// TwinCAT 3 PLC project Nepionic_Log_OTel
// Title: Nepionic_Log_OTel
// Company: Nepionic
// Author: Nepionic
// ProjectVersion: 0.1.0
// ProgramVersion: 3.1.4026.21
// libraries:
//   [Nepionic_Log], * (Nepionic)
//   Tc2_System, * (Beckhoff Automation GmbH)
//   Tc2_Utilities, * (Beckhoff Automation GmbH)
// project tree:
//   Lib/ OTelLogAppender.TcPOU, OTelLogEntry.TcDUT, OTelLogRing.TcDUT

// ---- Lib/OTelLogEntry.TcDUT
// One slot in the OTelLogRing.
//
// Binary layout (1280 bytes, little-endian, matches Go parser in adsbridge/ringbuf.go):
//
//   offset    0  ULINT   timestamp         Unix epoch nanoseconds
//   offset    8  UDINT   severity          0=Debug 1=Info 2=Warning 3=Error 4=Fatal
//   offset   12  UDINT   attr_count        Number of populated entries in attrs (0..10)
//   offset   16  BYTE[192] message         STRING(191) null-terminated
//   offset  208  BYTE[64]  source          STRING(63)  null-terminated (instance path)
//   offset  272  BYTE[960] attrs           ARRAY[0..9] OF LogAttribute (96 bytes each)
//                                            each attr:
//                                              offset  0  key         STRING(31)       = 32 bytes
//                                              offset 32  attr_type   LogAttributeType =  1 byte
//                                              offset 33  value_bytes ARRAY[0..62]     = 63 bytes
//   offset 1232  BYTE[44]  _pad
//   offset 1276  UDINT   sequence          ODD=being written, EVEN=committed (LAST field)
//   Total: 1280 bytes
{attribute 'pack_mode' := '1'}
TYPE OTelLogEntry :
STRUCT
	timestamp : ULINT;
	severity : UDINT;
	attribute_count : UDINT(0..10);
	message : STRING(191);
	source : STRING(63);
	attributes : ARRAY[0..9] OF Nepionic_Log.LogAttribute;
	_pad : ARRAY[0..43] OF BYTE;
	sequence : UDINT;
END_STRUCT
END_TYPE

// ---- Lib/OTelLogRing.TcDUT
// Ring buffer header + 128-slot log entry array.
// Exposed as an ADS symbol (e.g. OtelBridge.LogRing) and read by the Go collector.
//
// Binary layout:
//   offset  0  UDINT  head          Monotonically increasing write counter
//   offset  4  UDINT  capacity      Number of slots = 128
//   offset  8  UDINT  overflow_cnt  Incremented when ring is full
//   offset 12  UDINT  _reserved
//   offset 16  BYTE[48] _cache_pad  Pad header to 64 bytes
//   offset 64  OtelLogEntry[128]    128 × 1280 bytes = 163840 bytes
//   Total: 163904 bytes
TYPE OTelLogRing :
STRUCT
	head : UDINT;
	capacity : UDINT := 128;
	overflow_cnt : UDINT;
	_reserved : UDINT;
	_cache_pad : ARRAY[0..47] OF BYTE;
	entries : ARRAY[0..127] OF OTelLogEntry;
END_STRUCT
END_TYPE

// ---- Lib/OTelLogAppender.TcPOU
{attribute 'linkalways'}
{attribute 'no_explicit_call' := 'This FB is a CLASS and must be accessed using methods or properties'}
{attribute 'enable_dynamic_creation'}
/// OTel log appender for Nepionic_Log.
/// Implements `LogAppender` by writing structured log entries directly into its
/// own `OTelLogRing` field (`Ring`), which is exposed as an ADS symbol and
/// consumed by the Go `otelcol-ads` collector.
///
/// The ring is owned by the appender — no external ring declaration is needed.
/// Just declare the appender in a PROGRAM or GVL so TwinCAT generates an ADS
/// symbol for it, then point the collector at `<PROGRAM>.<var_name>.Ring`.
///
/// Usage:
/// ```st
/// // startup (e.g. MAIN FB_Init)
/// GetLogManager().Register(otel_appender);
///
/// // otelcol-ads config:
/// //   symbol: MAIN.otel_appender.Ring
/// ```
FUNCTION_BLOCK PUBLIC OTelLogAppender IMPLEMENTS Nepionic_Log.LogAppender
VAR
	{attribute 'otelcol_role' := 'log_ring'}
	ring : OTelLogRing;
	_level : Nepionic_Log.LogLevel := Nepionic_Log.LogLevel.Debug;
END_VAR

METHOD PUBLIC Append : BOOL
VAR_INPUT
	level : Nepionic_Log.LogLevel;
	message : Tc2_System.T_MaxString;
	source : Tc2_System.T_MaxString;
	attributes : ARRAY[0..9] OF Nepionic_Log.LogAttribute;
	attribute_count : USINT;
END_VAR
VAR
	slot_idx : UDINT;
	expected_gen : UDINT;
	file_time : ULINT;
	i : USINT;
END_VAR
slot_idx := ring.head MOD ring.capacity;
expected_gen := (ring.head / ring.capacity + 1) * 2;

// Mark slot as being written (ODD sequence = write in progress)
ring.entries[slot_idx].sequence := expected_gen - 1;

// Timestamp — Windows FILETIME → Unix nanoseconds
file_time := Tc2_Utilities.F_GetSystemTime();
ring.entries[slot_idx].timestamp := (file_time - 116444736000000000) * 100;

// Severity mapping
CASE level OF
	Nepionic_Log.LogLevel.Debug:
		ring.entries[slot_idx].severity := 0;
	Nepionic_Log.LogLevel.Information:
		ring.entries[slot_idx].severity := 1;
	Nepionic_Log.LogLevel.Warning:
		ring.entries[slot_idx].severity := 2;
	Nepionic_Log.LogLevel.Error:
		ring.entries[slot_idx].severity := 3;
	Nepionic_Log.LogLevel.Fatal:
		ring.entries[slot_idx].severity := 4;
ELSE
	ring.entries[slot_idx].severity := 1;
END_CASE

// Payload
ring.entries[slot_idx].message := message;
ring.entries[slot_idx].source := source;
ring.entries[slot_idx].attribute_count := USINT_TO_UDINT(attribute_count);
FOR i := 0 TO 9 DO
	ring.entries[slot_idx].attributes[i] := attributes[i];
END_FOR

// Commit slot (EVEN sequence = ready for reader)
ring.entries[slot_idx].sequence := expected_gen;

// Increment overflow counter each time the write pointer wraps back to slot 0.
IF slot_idx = 0 AND ring.head > 0 THEN
	ring.overflow_cnt := ring.overflow_cnt + 1;
END_IF

// Advance write cursor
ring.head := ring.head + 1;

Append := TRUE;
END_METHOD

{attribute 'monitoring' := 'call'}
PROPERTY PUBLIC Level : Nepionic_Log.LogLevel
GET // PUBLIC
Level := _level;
END_GET
SET // PUBLIC
_level := Level;
END_SET
END_PROPERTY

END_FUNCTION_BLOCK
